// TIA Portal V16 export
// export: Created 2024-09-05T15:58:42.8458985Z, ExportSetting WithDefaults, DisplayName Totally Integrated Automation Portal, DisplayVersion V16 Update 6, DisplayName TIA Portal Version Control Interface, DisplayVersion V16 Update 2, DisplayName TIA Portal Openness, DisplayVersion V16 Update 6, DisplayName STEP 7 Professional, DisplayVersion V16 Update 6, DisplayName STEP 7 Safety, DisplayVersion V16, DisplayName WinCC Advanced, DisplayVersion V16 Update 6
VAR_GLOBAL   // PLC tag table "DM_SM_LH"
   "DM_SMLH-TriggerEnable" AT %Q16.0 : Bool;
   "DM_SMLH-Trigger" AT %Q16.1 : Bool;
   "DM_SMLH-TriggerReady" AT %I32.0 : Bool;
   "DM_SMLH-TriggerAck" AT %I32.1 : Bool;
   "DM_SMLH-Acquiring" AT %I32.2 : Bool;
   "DM_SMLH-MissedAcq" AT %I32.3 : Bool;
   "DM_SMLH-TriggerID" AT %IW33 : Word;
   "DM_SMLH-BufferResultsEnable" AT %Q17.0 : Bool;
   "DM_SMLH-ResultsAck" AT %Q17.1 : Bool;
   "DM_SMLH-Decoding" AT %I36.0 : Bool;
   "DM_SMLH-Decode Complete" AT %I36.1 : Bool;
   "DM_SMLH-Results Buffer Overrun" AT %I36.2 : Bool;
   "DM_SMLH-Results Available" AT %I36.3 : Bool;
   "DM_SMLH-General Fault" AT %I36.7 : Bool;
   "DM_SMLH-Train Code" AT %Q18.0 : Bool;
   "DM_SMLH-Train Match String" AT %Q18.1 : Bool;
   "DM_SMLH-Train Focus" AT %Q18.2 : Bool;
   "DM_SMLH-Train Brightness" AT %Q18.3 : Bool;
   "DM_SMLH-Untrain" AT %Q18.4 : Bool;
   "DM_SMLH-Execute DMCC" AT %Q18.6 : Bool;
   "DM_SMLH-Set Match String" AT %Q18.7 : Bool;
   "DM_SMLH-Train Code Ack" AT %I37.0 : Bool;
   "DM_SMLH-Train Match String Ack" AT %I37.1 : Bool;
   "DM_SMLH-Train Focus Ack" AT %I37.2 : Bool;
   "DM_SMLH-Train Brightness Ack" AT %I37.3 : Bool;
   "DM_SMLH-Untrain Ack" AT %I37.4 : Bool;
   "DM_SMLH-Execute DMCC Ack" AT %I37.6 : Bool;
   "DM_SMLH-Set Match String Ack" AT %I37.7 : Bool;
   "DM_SMLH-UserData Option" AT %QW528 : Word;
   "DM_SMLH-UserData Length" AT %QW530 : Word;
   "DM_SMLH-UserData[0]" AT %QB532 : Byte;
   "DM_SMLH-UserData[1]" AT %QB533 : Byte;
   "DM_SMLH-UserData[2]" AT %QB534 : Byte;
   "DM_SMLH-UserData[3]" AT %QB535 : Byte;
   "DM_SMLH-UserData[4]" AT %QB536 : Byte;
   "DM_SMLH-UserData[5]" AT %QB537 : Byte;
   "DM_SMLH-UserData[6]" AT %QB538 : Byte;
   "DM_SMLH-UserData[7]" AT %QB539 : Byte;
   "DM_SMLH-UserData[8]" AT %QB540 : Byte;
   "DM_SMLH-UserData[9]" AT %QB541 : Byte;
   "DM_SMLH-UserData[10]" AT %QB542 : Byte;
   "DM_SMLH-UserData[11]" AT %QB543 : Byte;
   "DM_SMLH-UserData[12]" AT %QB544 : Byte;
   "DM_SMLH-UserData[13]" AT %QB545 : Byte;
   "DM_SMLH-UserData[14]" AT %QB546 : Byte;
   "DM_SMLH-UserData[15]" AT %QB547 : Byte;
   "DM_SMLH-ResultID" AT %IW600 : Word;
   "DM_SMLH-Result Code" AT %IW602 : Word;
   "DM_SMLH-Result Extended" AT %IW604 : Word;
   "DM_SMLH-Result Length" AT %IW606 : Word;
   "DM_SMLH-InspectionResults[0]" AT %IB608 : Byte;
   "DM_SMLH-InspectionResults[1]" AT %IB609 : Byte;
   "DM_SMLH-InspectionResults[2]" AT %IB610 : Byte;
   "DM_SMLH-InspectionResults[3]" AT %IB611 : Byte;
   "DM_SMLH-InspectionResults[4]" AT %IB612 : Byte;
   "DM_SMLH-InspectionResults[5]" AT %IB613 : Byte;
   "DM_SMLH-InspectionResults[6]" AT %IB614 : Byte;
   "DM_SMLH-InspectionResults[7]" AT %IB615 : Byte;
   "DM_SMLH-InspectionResults[8]" AT %IB616 : Byte;
   "DM_SMLH-InspectionResults[9]" AT %IB617 : Byte;
   "DM_SMLH-InspectionResults[10]" AT %IB618 : Byte;
   "DM_SMLH-InspectionResults[11]" AT %IB619 : Byte;
   "DM_SMLH-InspectionResults[12]" AT %IB620 : Byte;
   "DM_SMLH-InspectionResults[13]" AT %IB621 : Byte;
   "DM_SMLH-InspectionResults[14]" AT %IB622 : Byte;
   "DM_SMLH-InspectionResults[15]" AT %IB623 : Byte;
END_VAR
